// TIA Portal V17 export
// export: Created 2023-03-24T09:45:04.5136241Z, ExportSetting None, DisplayName Totally Integrated Automation Portal, DisplayVersion V17 Update 4, DisplayName TIA Portal Openness, DisplayVersion V17 Update 4, DisplayName TIA Portal Version Control Interface, DisplayVersion V17, DisplayName STEP 7 Professional, DisplayVersion V17 Update 4, DisplayName STEP 7 Safety, DisplayVersion V17, DisplayName WinCC Advanced / Unified PC, DisplayVersion V17 Update 4
FUNCTION "FC_DI" : Void   // FC12, LAD
TITLE = FC_DI
{ S7_Optimized_Access := 'FALSE' }
// Digital Input
// stored: SetENOAutomatically false
BEGIN

REGION Network 1: SOV EBV 33303 CLOSE FEEDBACK
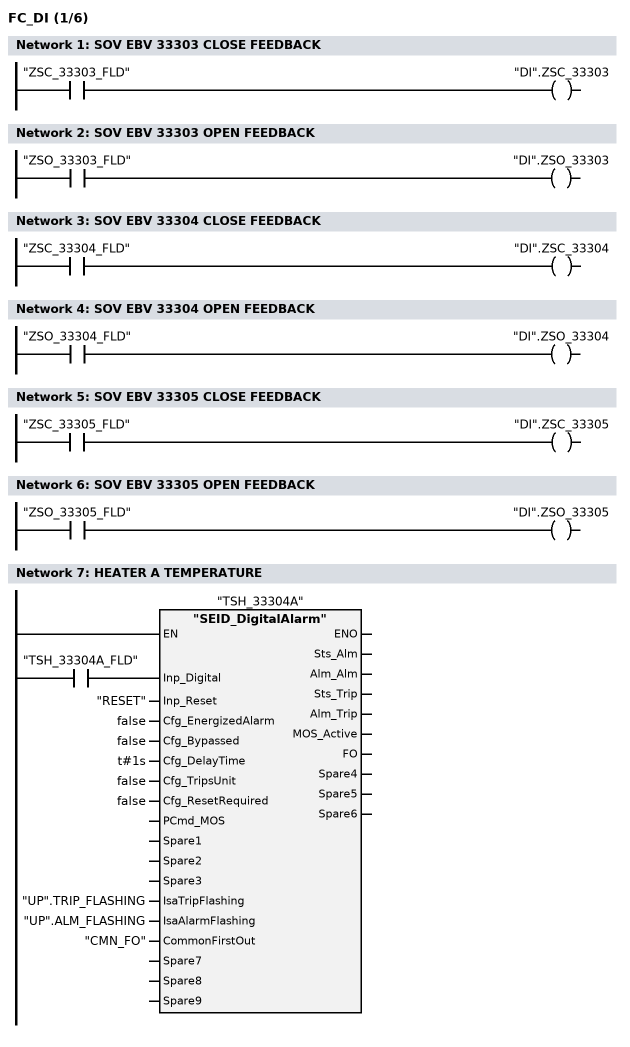
   RUNG wire#powerrail
      Contact( "ZSC_33303_FLD" )
      Coil( "DI".ZSC_33303 )
   END_RUNG
   // the same network as SCL:
   "DI".ZSC_33303 := "ZSC_33303_FLD";
END_REGION

REGION Network 2: SOV EBV 33303 OPEN FEEDBACK
   RUNG wire#powerrail
      Contact( "ZSO_33303_FLD" )
      Coil( "DI".ZSO_33303 )
   END_RUNG
   // the same network as SCL:
   "DI".ZSO_33303 := "ZSO_33303_FLD";
END_REGION

REGION Network 3: SOV EBV 33304 CLOSE FEEDBACK
   RUNG wire#powerrail
      Contact( "ZSC_33304_FLD" )
      Coil( "DI".ZSC_33304 )
   END_RUNG
   // the same network as SCL:
   "DI".ZSC_33304 := "ZSC_33304_FLD";
END_REGION

REGION Network 4: SOV EBV 33304 OPEN FEEDBACK
   RUNG wire#powerrail
      Contact( "ZSO_33304_FLD" )
      Coil( "DI".ZSO_33304 )
   END_RUNG
   // the same network as SCL:
   "DI".ZSO_33304 := "ZSO_33304_FLD";
END_REGION

REGION Network 5: SOV EBV 33305 CLOSE FEEDBACK
   RUNG wire#powerrail
      Contact( "ZSC_33305_FLD" )
      Coil( "DI".ZSC_33305 )
   END_RUNG
   // the same network as SCL:
   "DI".ZSC_33305 := "ZSC_33305_FLD";
END_REGION

REGION Network 6: SOV EBV 33305 OPEN FEEDBACK
   RUNG wire#powerrail
      Contact( "ZSO_33305_FLD" )
      Coil( "DI".ZSO_33305 )
   END_RUNG
   // the same network as SCL:
   "DI".ZSO_33305 := "ZSO_33305_FLD";
END_REGION

REGION Network 7: HEATER A TEMPERATURE
   RUNG wire#powerrail
      "TSH_33304A"(Inp_Digital := wire#w1, Inp_Reset := "RESET", Cfg_EnergizedAlarm := false, Cfg_Bypassed := false, Cfg_DelayTime := t#1s, Cfg_TripsUnit := false, Cfg_ResetRequired := false, PCmd_MOS :=, Spare1 :=, Spare2 :=, Spare3 :=, IsaTripFlashing := "UP".TRIP_FLASHING, IsaAlarmFlashing := "UP".ALM_FLASHING, CommonFirstOut := "CMN_FO", Spare7 :=, Spare8 :=, Spare9 :=, Sts_Alm =>, Alm_Alm =>, Sts_Trip =>, Alm_Trip =>, MOS_Active =>, FO =>, Spare4 =>, Spare5 =>, Spare6 =>)
   END_RUNG
   RUNG wire#powerrail
      Contact( "TSH_33304A_FLD" )
   END_RUNG wire#w1
   // the same network as SCL:
   "TSH_33304A"(Inp_Digital := "TSH_33304A_FLD",   // "SEID_DigitalAlarm"
                Inp_Reset := "RESET",
                Cfg_EnergizedAlarm := false,
                Cfg_Bypassed := false,
                Cfg_DelayTime := t#1s,
                Cfg_TripsUnit := false,
                Cfg_ResetRequired := false,
                IsaTripFlashing := "UP".TRIP_FLASHING,
                IsaAlarmFlashing := "UP".ALM_FLASHING,
                CommonFirstOut := "CMN_FO");
END_REGION

REGION Network 8: HEATER B TEMPERATURE
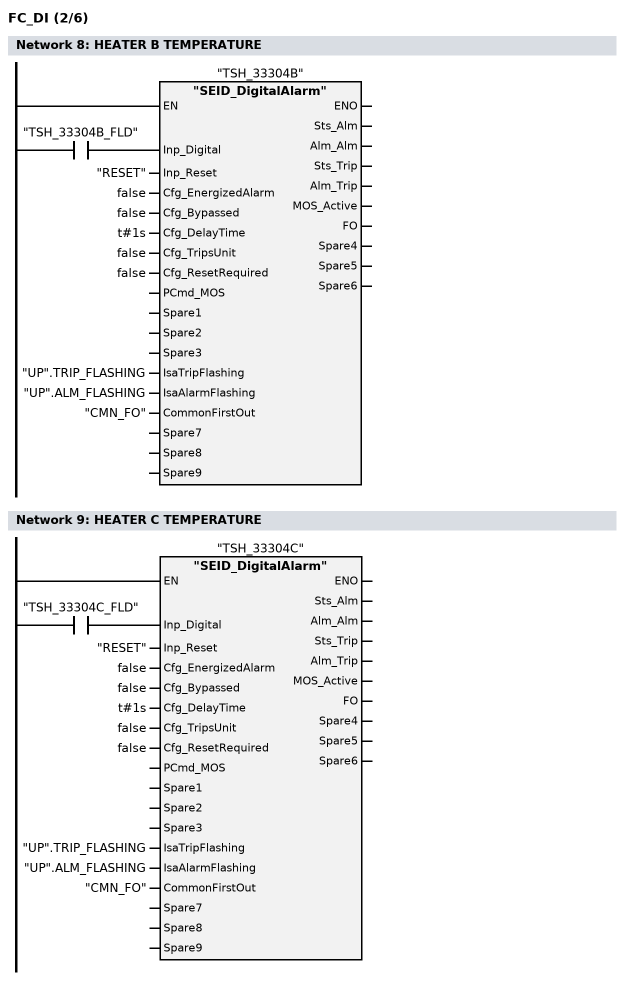
   RUNG wire#powerrail
      "TSH_33304B"(Inp_Digital := wire#w1, Inp_Reset := "RESET", Cfg_EnergizedAlarm := false, Cfg_Bypassed := false, Cfg_DelayTime := t#1s, Cfg_TripsUnit := false, Cfg_ResetRequired := false, PCmd_MOS :=, Spare1 :=, Spare2 :=, Spare3 :=, IsaTripFlashing := "UP".TRIP_FLASHING, IsaAlarmFlashing := "UP".ALM_FLASHING, CommonFirstOut := "CMN_FO", Spare7 :=, Spare8 :=, Spare9 :=, Sts_Alm =>, Alm_Alm =>, Sts_Trip =>, Alm_Trip =>, MOS_Active =>, FO =>, Spare4 =>, Spare5 =>, Spare6 =>)
   END_RUNG
   RUNG wire#powerrail
      Contact( "TSH_33304B_FLD" )
   END_RUNG wire#w1
   // the same network as SCL:
   "TSH_33304B"(Inp_Digital := "TSH_33304B_FLD",   // "SEID_DigitalAlarm"
                Inp_Reset := "RESET",
                Cfg_EnergizedAlarm := false,
                Cfg_Bypassed := false,
                Cfg_DelayTime := t#1s,
                Cfg_TripsUnit := false,
                Cfg_ResetRequired := false,
                IsaTripFlashing := "UP".TRIP_FLASHING,
                IsaAlarmFlashing := "UP".ALM_FLASHING,
                CommonFirstOut := "CMN_FO");
END_REGION

REGION Network 9: HEATER C TEMPERATURE
   RUNG wire#powerrail
      "TSH_33304C"(Inp_Digital := wire#w1, Inp_Reset := "RESET", Cfg_EnergizedAlarm := false, Cfg_Bypassed := false, Cfg_DelayTime := t#1s, Cfg_TripsUnit := false, Cfg_ResetRequired := false, PCmd_MOS :=, Spare1 :=, Spare2 :=, Spare3 :=, IsaTripFlashing := "UP".TRIP_FLASHING, IsaAlarmFlashing := "UP".ALM_FLASHING, CommonFirstOut := "CMN_FO", Spare7 :=, Spare8 :=, Spare9 :=, Sts_Alm =>, Alm_Alm =>, Sts_Trip =>, Alm_Trip =>, MOS_Active =>, FO =>, Spare4 =>, Spare5 =>, Spare6 =>)
   END_RUNG
   RUNG wire#powerrail
      Contact( "TSH_33304C_FLD" )
   END_RUNG wire#w1
   // the same network as SCL:
   "TSH_33304C"(Inp_Digital := "TSH_33304C_FLD",   // "SEID_DigitalAlarm"
                Inp_Reset := "RESET",
                Cfg_EnergizedAlarm := false,
                Cfg_Bypassed := false,
                Cfg_DelayTime := t#1s,
                Cfg_TripsUnit := false,
                Cfg_ResetRequired := false,
                IsaTripFlashing := "UP".TRIP_FLASHING,
                IsaAlarmFlashing := "UP".ALM_FLASHING,
                CommonFirstOut := "CMN_FO");
END_REGION

REGION Network 10: HEATER D TEMPERATURE
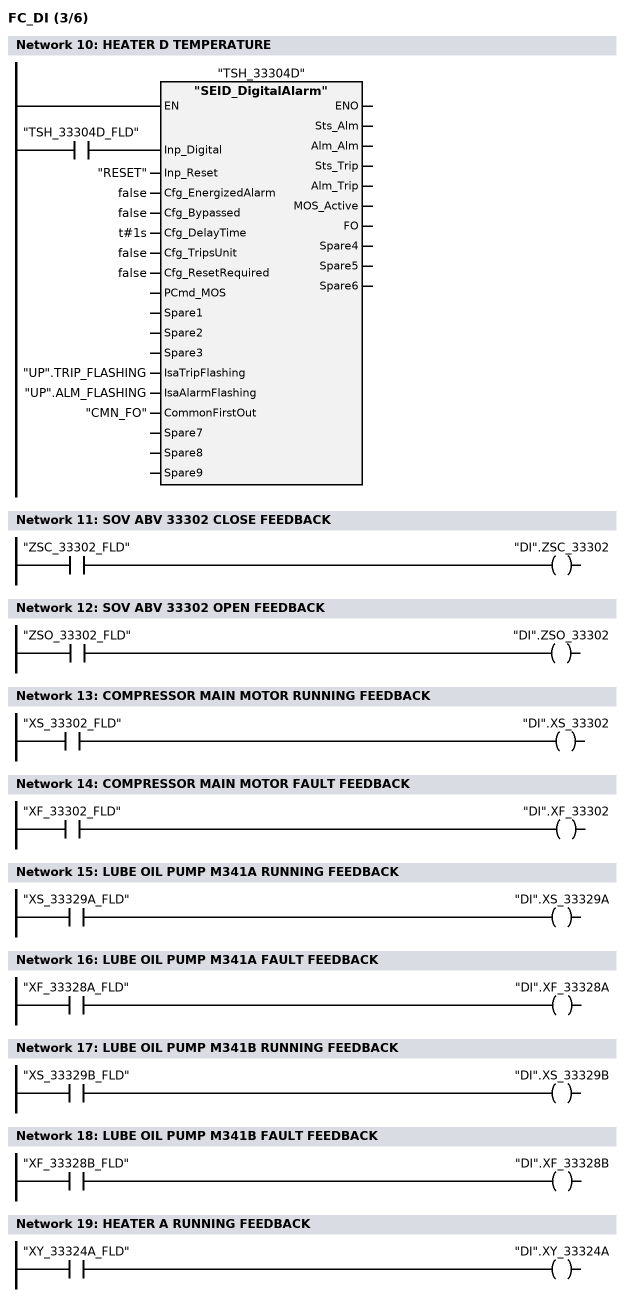
   RUNG wire#powerrail
      "TSH_33304D"(Inp_Digital := wire#w1, Inp_Reset := "RESET", Cfg_EnergizedAlarm := false, Cfg_Bypassed := false, Cfg_DelayTime := t#1s, Cfg_TripsUnit := false, Cfg_ResetRequired := false, PCmd_MOS :=, Spare1 :=, Spare2 :=, Spare3 :=, IsaTripFlashing := "UP".TRIP_FLASHING, IsaAlarmFlashing := "UP".ALM_FLASHING, CommonFirstOut := "CMN_FO", Spare7 :=, Spare8 :=, Spare9 :=, Sts_Alm =>, Alm_Alm =>, Sts_Trip =>, Alm_Trip =>, MOS_Active =>, FO =>, Spare4 =>, Spare5 =>, Spare6 =>)
   END_RUNG
   RUNG wire#powerrail
      Contact( "TSH_33304D_FLD" )
   END_RUNG wire#w1
   // the same network as SCL:
   "TSH_33304D"(Inp_Digital := "TSH_33304D_FLD",   // "SEID_DigitalAlarm"
                Inp_Reset := "RESET",
                Cfg_EnergizedAlarm := false,
                Cfg_Bypassed := false,
                Cfg_DelayTime := t#1s,
                Cfg_TripsUnit := false,
                Cfg_ResetRequired := false,
                IsaTripFlashing := "UP".TRIP_FLASHING,
                IsaAlarmFlashing := "UP".ALM_FLASHING,
                CommonFirstOut := "CMN_FO");
END_REGION

REGION Network 11: SOV ABV 33302 CLOSE FEEDBACK
   RUNG wire#powerrail
      Contact( "ZSC_33302_FLD" )
      Coil( "DI".ZSC_33302 )
   END_RUNG
   // the same network as SCL:
   "DI".ZSC_33302 := "ZSC_33302_FLD";
END_REGION

REGION Network 12: SOV ABV 33302 OPEN FEEDBACK
   RUNG wire#powerrail
      Contact( "ZSO_33302_FLD" )
      Coil( "DI".ZSO_33302 )
   END_RUNG
   // the same network as SCL:
   "DI".ZSO_33302 := "ZSO_33302_FLD";
END_REGION

REGION Network 13: COMPRESSOR MAIN MOTOR RUNNING FEEDBACK
   RUNG wire#powerrail
      Contact( "XS_33302_FLD" )
      Coil( "DI".XS_33302 )
   END_RUNG
   // the same network as SCL:
   "DI".XS_33302 := "XS_33302_FLD";
END_REGION

REGION Network 14: COMPRESSOR MAIN MOTOR FAULT FEEDBACK
   RUNG wire#powerrail
      Contact( "XF_33302_FLD" )
      Coil( "DI".XF_33302 )
   END_RUNG
   // the same network as SCL:
   "DI".XF_33302 := "XF_33302_FLD";
END_REGION

REGION Network 15: LUBE OIL PUMP M341A RUNNING FEEDBACK
   RUNG wire#powerrail
      Contact( "XS_33329A_FLD" )
      Coil( "DI".XS_33329A )
   END_RUNG
   // the same network as SCL:
   "DI".XS_33329A := "XS_33329A_FLD";
END_REGION

REGION Network 16: LUBE OIL PUMP M341A FAULT FEEDBACK
   RUNG wire#powerrail
      Contact( "XF_33328A_FLD" )
      Coil( "DI".XF_33328A )
   END_RUNG
   // the same network as SCL:
   "DI".XF_33328A := "XF_33328A_FLD";
END_REGION

REGION Network 17: LUBE OIL PUMP M341B RUNNING FEEDBACK
   RUNG wire#powerrail
      Contact( "XS_33329B_FLD" )
      Coil( "DI".XS_33329B )
   END_RUNG
   // the same network as SCL:
   "DI".XS_33329B := "XS_33329B_FLD";
END_REGION

REGION Network 18: LUBE OIL PUMP M341B FAULT FEEDBACK
   RUNG wire#powerrail
      Contact( "XF_33328B_FLD" )
      Coil( "DI".XF_33328B )
   END_RUNG
   // the same network as SCL:
   "DI".XF_33328B := "XF_33328B_FLD";
END_REGION

REGION Network 19: HEATER A RUNNING FEEDBACK
   RUNG wire#powerrail
      Contact( "XY_33324A_FLD" )
      Coil( "DI".XY_33324A )
   END_RUNG
   // the same network as SCL:
   "DI".XY_33324A := "XY_33324A_FLD";
END_REGION

REGION Network 20: HEATER A FAULT FEEDBACK
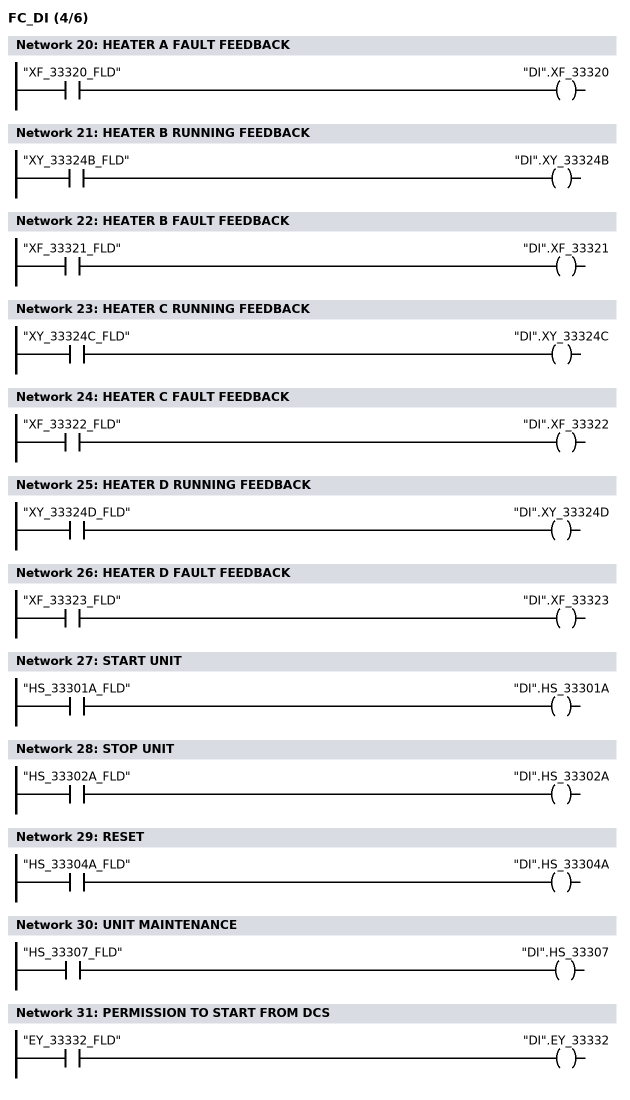
   RUNG wire#powerrail
      Contact( "XF_33320_FLD" )
      Coil( "DI".XF_33320 )
   END_RUNG
   // the same network as SCL:
   "DI".XF_33320 := "XF_33320_FLD";
END_REGION

REGION Network 21: HEATER B RUNNING FEEDBACK
   RUNG wire#powerrail
      Contact( "XY_33324B_FLD" )
      Coil( "DI".XY_33324B )
   END_RUNG
   // the same network as SCL:
   "DI".XY_33324B := "XY_33324B_FLD";
END_REGION

REGION Network 22: HEATER B FAULT FEEDBACK
   RUNG wire#powerrail
      Contact( "XF_33321_FLD" )
      Coil( "DI".XF_33321 )
   END_RUNG
   // the same network as SCL:
   "DI".XF_33321 := "XF_33321_FLD";
END_REGION

REGION Network 23: HEATER C RUNNING FEEDBACK
   RUNG wire#powerrail
      Contact( "XY_33324C_FLD" )
      Coil( "DI".XY_33324C )
   END_RUNG
   // the same network as SCL:
   "DI".XY_33324C := "XY_33324C_FLD";
END_REGION

REGION Network 24: HEATER C FAULT FEEDBACK
   RUNG wire#powerrail
      Contact( "XF_33322_FLD" )
      Coil( "DI".XF_33322 )
   END_RUNG
   // the same network as SCL:
   "DI".XF_33322 := "XF_33322_FLD";
END_REGION

REGION Network 25: HEATER D RUNNING FEEDBACK
   RUNG wire#powerrail
      Contact( "XY_33324D_FLD" )
      Coil( "DI".XY_33324D )
   END_RUNG
   // the same network as SCL:
   "DI".XY_33324D := "XY_33324D_FLD";
END_REGION

REGION Network 26: HEATER D FAULT FEEDBACK
   RUNG wire#powerrail
      Contact( "XF_33323_FLD" )
      Coil( "DI".XF_33323 )
   END_RUNG
   // the same network as SCL:
   "DI".XF_33323 := "XF_33323_FLD";
END_REGION

REGION Network 27: START UNIT
   RUNG wire#powerrail
      Contact( "HS_33301A_FLD" )
      Coil( "DI".HS_33301A )
   END_RUNG
   // the same network as SCL:
   "DI".HS_33301A := "HS_33301A_FLD";
END_REGION

REGION Network 28: STOP UNIT
   RUNG wire#powerrail
      Contact( "HS_33302A_FLD" )
      Coil( "DI".HS_33302A )
   END_RUNG
   // the same network as SCL:
   "DI".HS_33302A := "HS_33302A_FLD";
END_REGION

REGION Network 29: RESET
   RUNG wire#powerrail
      Contact( "HS_33304A_FLD" )
      Coil( "DI".HS_33304A )
   END_RUNG
   // the same network as SCL:
   "DI".HS_33304A := "HS_33304A_FLD";
END_REGION

REGION Network 30: UNIT MAINTENANCE
   RUNG wire#powerrail
      Contact( "HS_33307_FLD" )
      Coil( "DI".HS_33307 )
   END_RUNG
   // the same network as SCL:
   "DI".HS_33307 := "HS_33307_FLD";
END_REGION

REGION Network 31: PERMISSION TO START FROM DCS
   RUNG wire#powerrail
      Contact( "EY_33332_FLD" )
      Coil( "DI".EY_33332 )
   END_RUNG
   // the same network as SCL:
   "DI".EY_33332 := "EY_33332_FLD";
END_REGION

REGION Network 32: TRIP FROM DCS
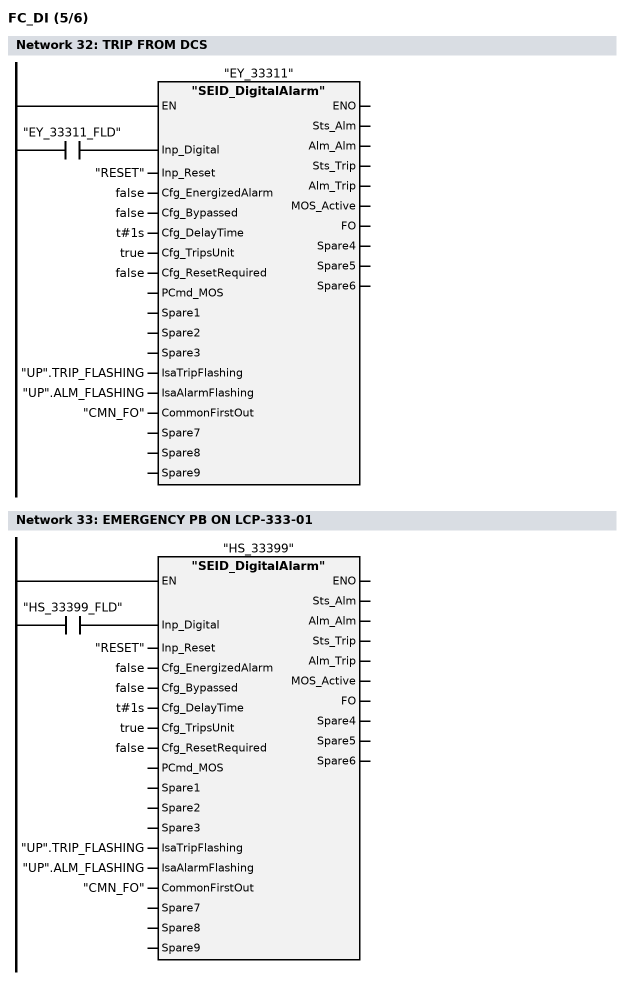
   RUNG wire#powerrail
      "EY_33311"(Inp_Digital := wire#w1, Inp_Reset := "RESET", Cfg_EnergizedAlarm := false, Cfg_Bypassed := false, Cfg_DelayTime := t#1s, Cfg_TripsUnit := true, Cfg_ResetRequired := false, PCmd_MOS :=, Spare1 :=, Spare2 :=, Spare3 :=, IsaTripFlashing := "UP".TRIP_FLASHING, IsaAlarmFlashing := "UP".ALM_FLASHING, CommonFirstOut := "CMN_FO", Spare7 :=, Spare8 :=, Spare9 :=, Sts_Alm =>, Alm_Alm =>, Sts_Trip =>, Alm_Trip =>, MOS_Active =>, FO =>, Spare4 =>, Spare5 =>, Spare6 =>)
   END_RUNG
   RUNG wire#powerrail
      Contact( "EY_33311_FLD" )
   END_RUNG wire#w1
   // the same network as SCL:
   "EY_33311"(Inp_Digital := "EY_33311_FLD",   // "SEID_DigitalAlarm"
              Inp_Reset := "RESET",
              Cfg_EnergizedAlarm := false,
              Cfg_Bypassed := false,
              Cfg_DelayTime := t#1s,
              Cfg_TripsUnit := true,
              Cfg_ResetRequired := false,
              IsaTripFlashing := "UP".TRIP_FLASHING,
              IsaAlarmFlashing := "UP".ALM_FLASHING,
              CommonFirstOut := "CMN_FO");
END_REGION

REGION Network 33: EMERGENCY PB ON LCP-333-01
   RUNG wire#powerrail
      "HS_33399"(Inp_Digital := wire#w1, Inp_Reset := "RESET", Cfg_EnergizedAlarm := false, Cfg_Bypassed := false, Cfg_DelayTime := t#1s, Cfg_TripsUnit := true, Cfg_ResetRequired := false, PCmd_MOS :=, Spare1 :=, Spare2 :=, Spare3 :=, IsaTripFlashing := "UP".TRIP_FLASHING, IsaAlarmFlashing := "UP".ALM_FLASHING, CommonFirstOut := "CMN_FO", Spare7 :=, Spare8 :=, Spare9 :=, Sts_Alm =>, Alm_Alm =>, Sts_Trip =>, Alm_Trip =>, MOS_Active =>, FO =>, Spare4 =>, Spare5 =>, Spare6 =>)
   END_RUNG
   RUNG wire#powerrail
      Contact( "HS_33399_FLD" )
   END_RUNG wire#w1
   // the same network as SCL:
   "HS_33399"(Inp_Digital := "HS_33399_FLD",   // "SEID_DigitalAlarm"
              Inp_Reset := "RESET",
              Cfg_EnergizedAlarm := false,
              Cfg_Bypassed := false,
              Cfg_DelayTime := t#1s,
              Cfg_TripsUnit := true,
              Cfg_ResetRequired := false,
              IsaTripFlashing := "UP".TRIP_FLASHING,
              IsaAlarmFlashing := "UP".ALM_FLASHING,
              CommonFirstOut := "CMN_FO");
END_REGION

REGION Network 34: LCP-333-01 INTERNAL HIGH TEMPERATURE
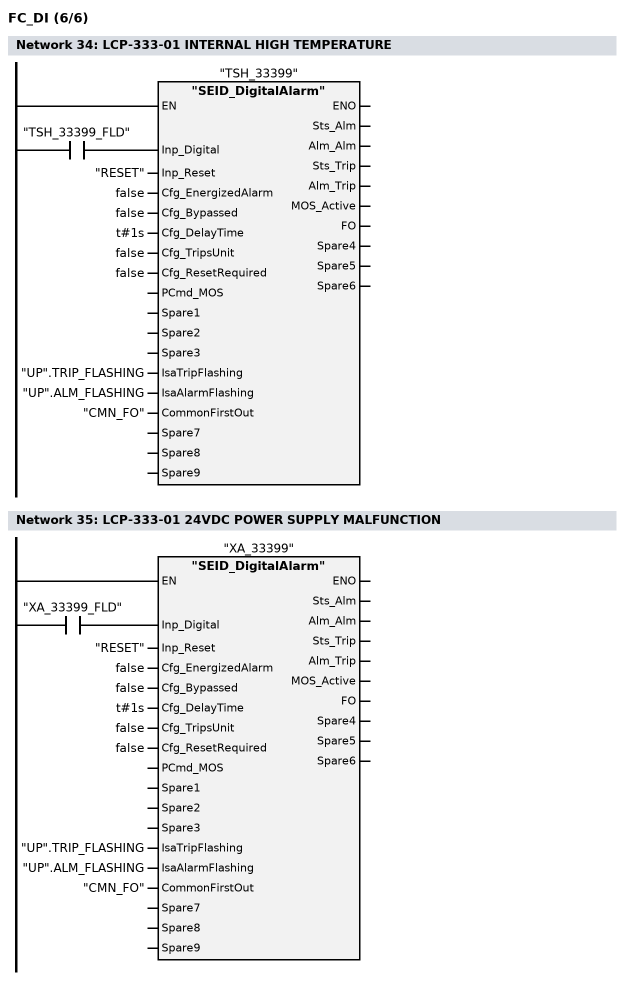
   RUNG wire#powerrail
      "TSH_33399"(Inp_Digital := wire#w1, Inp_Reset := "RESET", Cfg_EnergizedAlarm := false, Cfg_Bypassed := false, Cfg_DelayTime := t#1s, Cfg_TripsUnit := false, Cfg_ResetRequired := false, PCmd_MOS :=, Spare1 :=, Spare2 :=, Spare3 :=, IsaTripFlashing := "UP".TRIP_FLASHING, IsaAlarmFlashing := "UP".ALM_FLASHING, CommonFirstOut := "CMN_FO", Spare7 :=, Spare8 :=, Spare9 :=, Sts_Alm =>, Alm_Alm =>, Sts_Trip =>, Alm_Trip =>, MOS_Active =>, FO =>, Spare4 =>, Spare5 =>, Spare6 =>)
   END_RUNG
   RUNG wire#powerrail
      Contact( "TSH_33399_FLD" )
   END_RUNG wire#w1
   // the same network as SCL:
   "TSH_33399"(Inp_Digital := "TSH_33399_FLD",   // "SEID_DigitalAlarm"
               Inp_Reset := "RESET",
               Cfg_EnergizedAlarm := false,
               Cfg_Bypassed := false,
               Cfg_DelayTime := t#1s,
               Cfg_TripsUnit := false,
               Cfg_ResetRequired := false,
               IsaTripFlashing := "UP".TRIP_FLASHING,
               IsaAlarmFlashing := "UP".ALM_FLASHING,
               CommonFirstOut := "CMN_FO");
END_REGION

REGION Network 35: LCP-333-01 24VDC POWER SUPPLY MALFUNCTION
   RUNG wire#powerrail
      "XA_33399"(Inp_Digital := wire#w1, Inp_Reset := "RESET", Cfg_EnergizedAlarm := false, Cfg_Bypassed := false, Cfg_DelayTime := t#1s, Cfg_TripsUnit := false, Cfg_ResetRequired := false, PCmd_MOS :=, Spare1 :=, Spare2 :=, Spare3 :=, IsaTripFlashing := "UP".TRIP_FLASHING, IsaAlarmFlashing := "UP".ALM_FLASHING, CommonFirstOut := "CMN_FO", Spare7 :=, Spare8 :=, Spare9 :=, Sts_Alm =>, Alm_Alm =>, Sts_Trip =>, Alm_Trip =>, MOS_Active =>, FO =>, Spare4 =>, Spare5 =>, Spare6 =>)
   END_RUNG
   RUNG wire#powerrail
      Contact( "XA_33399_FLD" )
   END_RUNG wire#w1
   // the same network as SCL:
   "XA_33399"(Inp_Digital := "XA_33399_FLD",   // "SEID_DigitalAlarm"
              Inp_Reset := "RESET",
              Cfg_EnergizedAlarm := false,
              Cfg_Bypassed := false,
              Cfg_DelayTime := t#1s,
              Cfg_TripsUnit := false,
              Cfg_ResetRequired := false,
              IsaTripFlashing := "UP".TRIP_FLASHING,
              IsaAlarmFlashing := "UP".ALM_FLASHING,
              CommonFirstOut := "CMN_FO");
END_REGION
END_FUNCTION
